RoboDK station: project.rdk

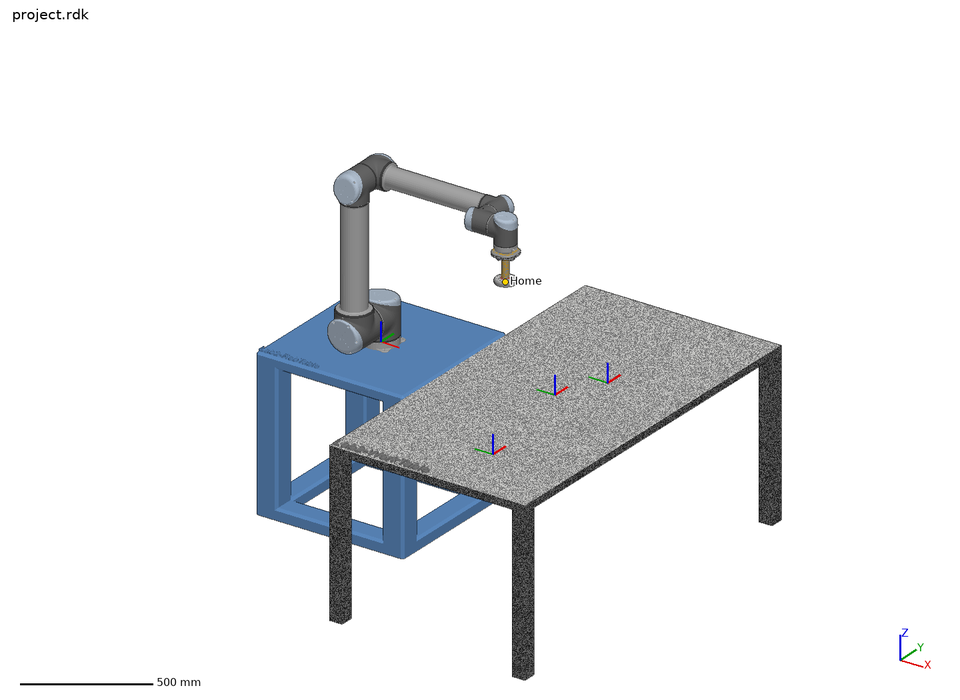
[picture v0: the station drawn from its stored meshes, robots at their saved joint values, targets as dots, program paths as lines]
Station project. Poses are relative to the parent item; angles as X-Y-Z fixed-axis rotations.
  - frame roboBase at (0, 1000, 0) mm
    - robot robot: 6 axes, payload 10 kg, reach 1300 mm, repeatability 0.1 mm, weight 28.9 kg
        modified DH rows (alpha deg, a mm, theta deg, d mm): 0, 0, 0, 118; 90, 0, 180, 0; 0, 612.7, 0, 0; 0, 571.6, 0, 163.9; -90, 0, 0, 115.7; 90, 0, 180, 92.2
        joint limits [-360, -360, -360, -360, -360, -360] to [360, 360, 360, 360, 360, 360]; home [0, -90, -90, 0, 90, 0]; saved at [0, -90, -90, -90, 90, 0]
      - tool tool, TCP at (0, 0, 130) mm, size 100 x 100 x 133.5 mm, geometry from CostumTool.iges
    - object RobTable at (0, 0, 0) mm, size 680 x 680 x 690 mm, geometry from RobTable.iges
    - target Home (Cartesian target) at (687.3, -163.9, 508.5) mm, rotated rx 180 ry 0 rz -90 deg; joints [0, -90, -90, -90, 90, 0] of robot
    - frame pickFrame at (800, 0, 0) mm, rotated rx 0 ry 0 rz 90 deg
      - frame placeFrameLeft at (-550, -100, 0) mm
      - frame placeFrameRight at (200, -100, 0) mm
    - object WorkTable at (800, 0, 0) mm, size 900 x 1680 x 742 mm, geometry from WorkTable.iges
